(* IEC 61131-3 sources: Heukranen/, 1 file *)

(* ---- my_struct.st ---- *)
VAR
  array: ARRAY [a, b, c] OF INT;
END_VAR
